(* CODESYS project tc_collections.library
   Company: Red Rock Controls
   Version: 1.0.0.8
   Description: RemoveLast() added
      TIniFile added
   Author: Roger Christopher
   Title: Tc_Collections

Project tree, tasks and I/O mapping:
  libraries: Tc2_Standard, * (Beckhoff Automation GmbH); Tc2_System, * (Beckhoff Automation GmbH); Tc2_Utilities, * (Beckhoff Automation GmbH); Tc_Helper, 1.0.0.5 (Red Rock Controls)
  Collections/
    Ini File/
      data type TIniEntry
      function block TIniFile [ST]: AddEntry, AddSection, GetValue, IniEntryToString, SetValue, StringToIniEntry
    String List/
      function block FB_ReadStringListFromFile [ST]
      function block FB_WriteStringListToFile [ST]
      data type TReadFromFile_State
      function block TStringIterator [ST]: GetCurrent, Index, Init, MoveNext
      function block TStringList [ST]: AddItem, Clear, Count, Full, GetItem, InsertItem, RemoveItem, RemoveLast, SetItem
      data type TWriteToFile_State
  Version/
    global variables Global_Version
*)

// Collections/Ini File/TIniEntry
TYPE TIniEntry :
STRUCT
	Section: STRING;
	Name: STRING;
	Value: STRING;
	Comment: STRING;
END_STRUCT
END_TYPE

// Collections/String List/TReadFromFile_State
TYPE TReadFromFile_State :
(
	sInit,
	sOpenFile,
	sReadFile,
	sCloseFile,
	sError
);
END_TYPE

// Collections/String List/TWriteToFile_State
TYPE TWriteToFile_State :
(
	sInit,
	sOpenFile,
	sWriteFile,
	sCloseFile,
	sError
);
END_TYPE

// Version/Global_Version
// This function has been automatically generated from the project information.
VAR_GLOBAL CONSTANT
	{attribute 'const_non_replaced'}
	stLibVersion_Tc_Collections : ST_LibVersion := (iMajor := 1, iMinor := 0, iBuild := 0, iRevision := 8, sVersion := '1.0.0.8');
END_VAR

// Collections/Ini File/TIniFile
FUNCTION_BLOCK TIniFile EXTENDS TStringList
VAR CONSTANT
	INI_COMMENT_DELIMITTER: STRING(1) := ';';
END_VAR

METHOD AddEntry : BOOL
VAR_INPUT
	Name: STRING;
	Value: STRING;
	Comment: STRING;
END_VAR
VAR
	IniEntry: TIniEntry;
END_VAR
(*Add ini file entry*)
IniEntry.Section := '';
IniEntry.Name := Name;
IniEntry.Comment := Comment;
IniEntry.Value := Value;
AddItem(In := IniEntryToString(IniEntry));
END_METHOD

METHOD AddSection : BOOL
VAR_INPUT
	Section: STRING;
END_VAR
VAR
	IniEntry: TIniEntry;
END_VAR
IniEntry.Section := Section;
IniEntry.Name := '';
IniEntry.Comment := '';
IniEntry.Value := '';
AddItem(In := IniEntryToString(IniEntry));
END_METHOD

METHOD GetValue : T_MaxString
VAR_INPUT
	Section: STRING;
	Name: STRING;
END_VAR
VAR
	Iterator: TStringIterator;
	CurrentSection: STRING;
	IniEntry: TIniEntry;
    i : INT;
END_VAR
GetValue := F_Concat6(
						s1 := 'Value not found. Section = "',
						s2 := Section,
						s3 := '", Name = "',
						s4 := Name,
						s5 := '"',
						s6 := '');
                        
FOR i := 0 TO _Count DO
 	IniEntry := StringToIniEntry(_Items[i]);
	IF IniEntry.Section <> '' THEN (*Just entered a new section*)
		CurrentSection := IniEntry.Section;
	END_IF
	IF CurrentSection = Section THEN (*We are in the required section*)
		IF IniEntry.Name = Name THEN
			GetValue := IniEntry.Value;
			RETURN;
		END_IF
	END_IF
END_FOR
END_METHOD

METHOD IniEntryToString : T_MaxString
VAR_INPUT
	IniEntry: TIniEntry;
END_VAR
VAR
	Result: T_MaxString;
END_VAR
IF IniEntry.Section <> '' AND (IniEntry.Name = '') THEN (*Entry should be either a section or a value, not both*)
	(*Write the formatted section*)
	Result:= F_Concat4(
						s1 := '[',
						s2 := IniEntry.Section,
						s3 := ']',
						s4 := '');
ELSIF (IniEntry.Name <> '') THEN
	(*Write the name/value pair*)
	Result:= F_Concat4(
						s1 := '  ',
						s2 := IniEntry.Name,
						s3 := ' = ',
						s4 := IniEntry.Value);
END_IF

(*Add comment. if any*)
IF IniEntry.Comment = '' THEN
	(*Just append an end-of-line character*)
	Result:= F_Concat2(
						s1 := Result,
						s2 := '$N');
ELSE
	(*Append comment and end-of-line*)
	Result:= F_Concat6(
						s1 := Result,
						s2 := INI_COMMENT_DELIMITTER,
						s3 := ' ',
						s4 := IniEntry.Comment,
						s5 := '$N',
						s6 := '');
END_IF

IniEntryToString := Result;
END_METHOD

METHOD SetValue : BOOL
VAR_INPUT
	Section: STRING;
	Name: STRING;
	Value: STRING;
	Comment: STRING;
END_VAR
VAR
	Iterator: TStringIterator;
	Line: T_MaxString;
	CurrentSection: STRING;
	IniEntry: TIniEntry;
	SectionFound: BOOL;
    i : INT;
END_VAR
FOR i := 0 TO _Count DO
 	IniEntry := StringToIniEntry(_Items[i]);
	IF IniEntry.Section <> '' THEN (*Just entered a new section*)
		CurrentSection := IniEntry.Section;
	END_IF
	IF CurrentSection = Section THEN (*We are in the required section*)
			SectionFound := TRUE;
			IF IniEntry.Name = Name THEN
				(*Update value*)
				IniEntry.Value := Value;
				IniEntry.Comment := Comment;
				Line := IniEntryToString(IniEntry);
				SetItem(Index := i, In := Line);
				SetValue := TRUE;
				RETURN;
			END_IF
	END_IF
END_FOR


(*Entry with required Section and Name not found, so add it to IniFile*)
IF NOT SectionFound THEN (*Add Section entry*)
	IniEntry.Section := Section;
	IniEntry.Name := '';
	IniEntry.Comment := '';
	IniEntry.Value := '';
	AddItem(In := IniEntryToString(IniEntry));
END_IF

(*Add ini file entry*)
IniEntry.Section := '';
IniEntry.Name := Name;
IniEntry.Comment := Comment;
IniEntry.Value := Value;
AddItem(In := IniEntryToString(IniEntry));
END_METHOD

METHOD StringToIniEntry : TIniEntry
VAR_INPUT
	Line: STRING;
END_VAR
VAR
	///Position of '['
	p1: INT;
	///Position of ']'
	p2: INT;
	///Position of '='
	p3: INT;
	///Position of comment delimiter
	p4: INT;
	///Position of end of line
	p5: INT;
	Length: INT;
	Result: TIniEntry;
END_VAR
(* Find section name in [SectionName] ; etc *)

p1 := FIND(Line,'[');
p2 := FIND(Line,']');

Length := p2 - p1 - 1;
IF (p1 > 0) AND (p2 > 0) AND (Length > 0) THEN
	Result.Section := F_Trim(MID(Line,Length,p1+1));
END_IF

p3 := FIND(Line,'=');
p4 := FIND(Line,INI_COMMENT_DELIMITTER);
p5 := FIND(Line,'$R');
IF p5 = 0 THEN
	p5 := FIND(Line,'$N');
END_IF
IF p5 = 0 THEN
	p5 := LEN(Line);
END_IF

(*Get name*)
IF (p1 = 0) AND (p2 = 0) AND (p3 > 0) THEN
	Result.Name := F_Trim(LEFT(Line, p3-1));
END_IF

(*Get value*)
IF (p3 > 0) AND (Result.Name <> '') THEN
	IF p4 = 0 THEN (* comment delimitter not found - use all remainder of string*)
		Length := p5 - p3 - 1;
	ELSE
		Length := p4 - p3 - 1;
	END_IF
	Result.Value := F_Trim(MID(Line,Length,p3+1));
END_IF

(*Get comment*)
IF p4 > 0 THEN
	Length := p5 - p4 - 1;
	Result.Comment := F_Trim(MID(Line,Length,p4+1));
END_IF

StringToIniEntry := Result;
END_METHOD

END_FUNCTION_BLOCK

// Collections/String List/TStringList
FUNCTION_BLOCK TStringList
VAR
	_Count: INT;
	_Items: ARRAY[0..MAX_LIST_ENTRIES-1] OF T_MaxString;
END_VAR
VAR CONSTANT
	MAX_LIST_ENTRIES: INT := 100;
END_VAR

;

METHOD AddItem : BOOL
VAR_INPUT
	In: T_MaxString;
END_VAR
IF NOT Full THEN
	_Items[Count] := In;
	_Count := _Count + 1;
END_IF
END_METHOD

METHOD Clear
VAR_INPUT
END_VAR
MEMSET(destAddr := ADR(_Items), fillByte := 0, n := SIZEOF(_Items));
_Count := 0;
END_METHOD

PROPERTY Count : INT
GET
Count := _Count;
END_GET
END_PROPERTY

PROPERTY Full : BOOL
GET
Full := (_Count >= MAX_LIST_ENTRIES);
END_GET
END_PROPERTY

METHOD GetItem : T_MaxString
VAR_INPUT
	Index : INT;// zero based
END_VAR
IF Index >= 0 AND Index < _Count THEN
	GetItem := _Items[Index];
END_IF
END_METHOD

METHOD InsertItem
VAR_INPUT
	In: T_MaxString;
END_VAR
IF NOT Full THEN
    MEMMOVE(destAddr := ADR(_Items[1]),
            srcAddr  := ADR(_Items[0]),
            n        := INT_TO_UINT(_Count) * SIZEOF(_Items[0]));

	_Items[0] := In;
	_Count := _Count + 1;
END_IF
END_METHOD

METHOD RemoveItem
VAR_INPUT
    Index : INT;//zero based
END_VAR
VAR
    NoItemsToMove : UINT;
END_VAR
IF _Count > 0 AND Index >= 0 THEN
    NoItemsToMove := INT_TO_UINT(_Count - Index - 1);  // if we have 4 items and want to remove item at index 1(zero based) we must move 4-1-1 items up
    IF NoItemsToMove > 0 THEN
        // shuffle items up in list
        MEMMOVE(destAddr:= ADR(_Items[Index]), 
                srcAddr:= ADR(_Items[Index + 1]), 
                n:= NoItemsToMove * SIZEOF(_Items[0]));
                
        // clear initialse freed up space
        MEMSET(destAddr:= ADR(_Items[_Count-1]),
               fillByte:= 0,
               n := SIZEOF(_Items[0]));

        _Count := _Count - 1;
        
    ELSIF NoItemsToMove = 0 THEN // removing last item 

        // initialise freed up space
        MEMSET(destAddr:= ADR(_Items[_Count-1]),
               fillByte:= 0,
               n := SIZEOF(_Items[0]));
    
        _Count := _Count - 1;
    END_IF
END_IF
END_METHOD

METHOD RemoveLast
IF _Count > 0 THEN          // last item exists
    MEMSET(destAddr := ADR(_Items[_Count-1]),
           fillByte := 0,
           n        := SIZEOF(_Items[0]));
    _Count := _Count - 1;   // update count
END_IF
END_METHOD

METHOD SetItem
VAR_INPUT
	In: T_MaxString;
	Index : INT;//zero based
END_VAR
IF Index < _Count AND Index > 0 THEN
	_Items[Index] := In;
END_IF
END_METHOD

END_FUNCTION_BLOCK

// Collections/String List/TStringIterator
FUNCTION_BLOCK TStringIterator
VAR
	_Index: INT;
	_List : REFERENCE TO TStringList;
END_VAR

METHOD GetCurrent : T_MaxString;
VAR_INPUT
END_VAR
GetCurrent := _List.GetItem(_Index);
END_METHOD

PROPERTY Index : INT
GET
Index := _Index;
END_GET
END_PROPERTY

METHOD Init
VAR_INPUT
	List : REFERENCE TO TStringList;
END_VAR
// set ref to StringList
_List REF= List;

// Initialise the current record pointer
_Index := -1;
END_METHOD

METHOD MoveNext : BOOL
VAR_INPUT
END_VAR
MoveNext := _List.Count >= 0 AND _Index < _List.Count;
IF MoveNext THEN
	_Index := _Index + 1;
END_IF
END_METHOD

END_FUNCTION_BLOCK

// Collections/String List/FB_ReadStringListFromFile
FUNCTION_BLOCK FB_ReadStringListFromFile
VAR_INPUT
	Execute: BOOL;
	AmsNetId : STRING(23);
	Path: T_MaxString;
END_VAR
VAR_IN_OUT
	StringList: TStringList;
END_VAR
VAR_OUTPUT
	Done: BOOL;
	Busy: BOOL;
	Error: BOOL;
	ErrorID: UDINT;
END_VAR
VAR
	State: TReadFromFile_State;
	Timeout: TIME := TIME#4s0ms;
	hFile: UINT;
	Line: T_MaxString;
	EOF: BOOL;
	R_TRIG1: R_TRIG;
	ExecuteRisingEdge: BOOL;
	FB_FileOpen1: FB_FileOpen;
	FB_FileGets1: FB_FileGets;
	FB_FileClose1: FB_FileClose;
	fbBusy: BOOL;
END_VAR

R_TRIG1(CLK:= Execute, Q=> ExecuteRisingEdge);
CASE State OF
	TReadFromFile_State.sInit:
		Busy := FALSE;
		IF ExecuteRisingEdge THEN
			Busy := TRUE;
			Done := FALSE;
			Error := FALSE;
			ErrorID := 0;
			State := TReadFromFile_State.sOpenFile;
			StringList.Clear();
		END_IF

	TReadFromFile_State.sOpenFile:
		FB_FileOpen1(
			sNetId:= AmsNetId,
			sPathName:= Path,
			nMode:= FOPEN_MODEREAD OR FOPEN_MODETEXT,
			ePath:= PATH_GENERIC,
			bExecute:= TRUE,
			tTimeout:= Timeout,
			bError=> Error,
			nErrID=> ErrorID,
			hFile=> hFile);
		IF NOT FB_FileOpen1.bBusy THEN
			IF NOT Error THEN
				State := TReadFromFile_State.sReadFile;
			ELSE
				State := TReadFromFile_State.sInit;
			END_IF
			FB_FileOpen1(bExecute := FALSE);
		END_IF

	TReadFromFile_State.sReadFile:
		FB_FileGets1(
			sNetId:= AmsNetId,
			hFile:= hFile,
			bExecute:= TRUE,
			tTimeout:= Timeout,
			bError=> Error,
			nErrId=> ErrorID,
			sLine=> Line,
			bEOF=> EOF);

		IF NOT FB_FileGets1.bBusy THEN
			FB_FileGets1(bExecute := FALSE);
			IF Error OR EOF  THEN
				State := TReadFromFile_State.sCloseFile;
			ELSE
				IF NOT StringList.Full THEN
					StringList.AddItem(In := Line);
				ELSE
					Error := TRUE;
					ErrorId := 100;
					State := TReadFromFile_State.sCloseFile;
				END_IF
			END_IF
		END_IF

	TReadFromFile_State.sCloseFile:
		FB_FileClose1(
			sNetId:= AmsNetId,
			hFile:= hFile,
			bExecute:= TRUE,
			tTimeout:= Timeout);
		IF NOT FB_FileClose1.bBusy THEN
			FB_FileClose1(bExecute := FALSE);
			Done := TRUE;
			Busy := FALSE;
			State := TReadFromFile_State.sInit;
		END_IF
END_CASE

END_FUNCTION_BLOCK

// Collections/String List/FB_WriteStringListToFile
FUNCTION_BLOCK FB_WriteStringListToFile
VAR_INPUT
	Execute: BOOL;
	AmsNetId : STRING(23);
	Path: T_MaxString;
END_VAR
VAR_IN_OUT
	StringList: TStringList;
END_VAR
VAR_OUTPUT
	Done: BOOL;
	Busy: BOOL;
	Error: BOOL;
	ErrorID: UDINT;
END_VAR
VAR
	State: TWriteToFile_State;
	Timeout: TIME := TIME#1s0ms;
	Iterator: TStringIterator;
	hFile: UINT;
	R_TRIG1: R_TRIG;
	ExecuteRisingEdge: BOOL;
	Line : T_MaxString;
	FB_FileOpen1: FB_FileOpen;
	FB_FilePuts1: FB_FilePuts;
	FB_FileClose1: FB_FileClose;
END_VAR

R_TRIG1(CLK:= Execute, Q=> ExecuteRisingEdge);
CASE State OF
	TWriteToFile_State.sInit:
		Busy := FALSE;
		IF ExecuteRisingEdge THEN
			Iterator.Init(StringList);
			IF Iterator.MoveNext() THEN (*We have entries to write...*)
				Busy := TRUE;
				Done := FALSE;
				Error := FALSE;
				ErrorID := 0;
				State := TWriteToFile_State.sOpenFile;
			END_IF
		END_IF

	TWriteToFile_State.sOpenFile:
		FB_FileOpen1(
			sNetId:= AmsNetId,
			sPathName:= Path,
			nMode:= FOPEN_MODEWRITE OR FOPEN_MODETEXT,
			ePath:= PATH_GENERIC,
			bExecute:= TRUE,
			tTimeout:= Timeout,
			bError=> Error,
			nErrID=> ErrorID,
			hFile=> hFile);
		IF NOT FB_FileOpen1.bBusy THEN
			IF NOT Error THEN
				Line := Iterator.GetCurrent();
				State := TWriteToFile_State.sWriteFile;
			ELSE
				State := TWriteToFile_State.sInit;
			END_IF
			FB_FileOpen1(bExecute := FALSE);
		END_IF

	TWriteToFile_State.sWriteFile:

		FB_FilePuts1(
			sNetId:= AmsNetId,
			hFile:= hFile,
			sLine:= Line,
			bExecute:= TRUE,
			tTimeout:= Timeout,
			bBusy=> ,
			bError=> Error,
			nErrId=> ErrorId);

		IF NOT FB_FilePuts1.bBusy THEN
			FB_FilePuts1(bExecute := FALSE);
			IF Error THEN
				State := TWriteToFile_State.sCloseFile;
			ELSE
				IF Iterator.MoveNext()  THEN 
					Line := Iterator.GetCurrent();
				ELSE (*Done*)
					State := TWriteToFile_State.sCloseFile;
				END_IF
			END_IF
		END_IF

	TWriteToFile_State.sCloseFile:
		FB_FileClose1(
			sNetId:= AmsNetId,
			hFile:= hFile,
			bExecute:= TRUE,
			tTimeout:= Timeout);
		IF NOT FB_FileClose1.bBusy THEN
			FB_FileClose1(bExecute := FALSE);
			Done := TRUE;
			Busy := FALSE;
			State := TWriteToFile_State.sInit;
		END_IF
END_CASE

END_FUNCTION_BLOCK
